FUNCTION_BLOCK SmallSortingConveyor EXTENDS Conveyor
VAR_INPUT
END_VAR
VAR_OUTPUT
END_VAR
VAR
	//Sensors
	m_PresencesensorStart : PresenceSensor;
	m_PresencesensorEnd : PresenceSensor;
	m_Opticalsensor : OpticalSensor;
	m_Inductivesensor : InductiveSensor;
	
	//Ramps
	m_Ramp : Ramp;
	
	//Pusher
	m_Switch : Switch;
END_VAR

PROPERTY LightWPAtMid : BOOL
GET
LightWPAtMid := m_Opticalsensor.Value;
END_GET
END_PROPERTY

PROPERTY MetalWPAtMid : BOOL
GET
MetalWPAtMid := m_Inductivesensor.Value;
END_GET
END_PROPERTY

METHOD METH_Switch_Extend : BOOL
VAR_INPUT
END_VAR
m_Switch.METH_Extend();
END_METHOD

METHOD METH_Switch_Retract : BOOL
VAR_INPUT
END_VAR
m_Switch.METH_Retract();
END_METHOD

PROPERTY WPAtEnd : BOOL
GET
WPAtEnd := m_PresencesensorEnd.Value;
END_GET
END_PROPERTY

PROPERTY WPAtRampEnd : BOOL
GET
WPAtRampEnd := m_Ramp.m_presenceSensorRampFull.Value;
END_GET
END_PROPERTY

PROPERTY WPAtStart : BOOL
GET
WPAtStart := m_PresencesensorStart.Value;
END_GET
END_PROPERTY

END_FUNCTION_BLOCK

(* stored: Version 1.1.0.1
   POU SmallSortingConveyor: Id {2a6136f6-689d-4559-bac8-e4f193940053}, SpecialFunc None
   Folder Methods: Id {6af266dd-85b9-41ba-a513-da971bc585a6}
   Folder Properties: Id {b8675340-e3ff-44e3-a956-05c73051eb9b}
   Property LightWPAtMid: Id {9f86efd5-82e6-44ca-ad22-72488d99bbdd}
   Get Get: Id {889a71e2-3cf0-434e-acf3-54b8161df2b8}
   Property MetalWPAtMid: Id {0b15feab-d48b-4e21-b4ea-5e5a7bd49c6f}
   Get Get: Id {db08b0b8-80bd-4681-8fdb-7fabc57de5c2}
   Method METH_Switch_Extend: Id {9a88a623-f65c-4520-95af-303d87e1dcd4}
   Method METH_Switch_Retract: Id {7d5e5f58-11a5-4799-9210-0090cb98a83b}
   Property WPAtEnd: Id {d4b30ce1-0d5a-41c1-887b-12cc4a5ce376}
   Get Get: Id {db781fcc-af48-449d-86fe-60e3c444eb04}
   Property WPAtRampEnd: Id {4161c70e-fd51-466d-ad67-93ac69901cab}
   Get Get: Id {0cc2b0f4-3950-41c1-ade7-56af5066394e}
   Property WPAtStart: Id {09f83741-4ba9-4fa1-8fe6-c28b540a671c}
   Get Get: Id {d3942da8-86bb-4efa-96d6-e07c398db4e0} *)
